// TIA Portal project "Endüstriyel Kapı" (V17)

(* hardware
DEVICE "S71500/ET200MP-Station_1"  S7-1500 station
   slot 0: "Profilschiene_0"  6ES7 590-1***0-0AA0
   slot 1: "PLC_1"  CPU 1511-1 PN  6ES7 511-1AK00-0AB0  V1.8
   slot 2: "AI 8xU/I/RTD/TC ST_1"  AI 8xU/I/RTD/TC ST  6ES7 531-7KF00-0AB0  V2.0
   slot 3: "AI 8xU/I/RTD/TC ST_2"  AI 8xU/I/RTD/TC ST  6ES7 531-7KF00-0AB0  V2.0
   slot 4: "AI 8xU/I/RTD/TC ST_3"  AI 8xU/I/RTD/TC ST  6ES7 531-7KF00-0AB0  V2.0
   slot 5: "AI 8xU/I/RTD/TC ST_4"  AI 8xU/I/RTD/TC ST  6ES7 531-7KF00-0AB0  V2.0
   slot 6: "DI 16x24VDC BA_1"  DI 16x24VDC BA  6ES7 521-1BH10-0AA0  V1.0
*)

// ===== PLC "PLC_1"  CPU 1511-1 PN =====

VAR_GLOBAL   // PLC tag table "Standard-Variablentabelle"
   "AÇMA (MÜHÜRLÜ)" AT %E0.0 : Bool;
   "AÇMA (KESİK)" AT %E0.1 : Bool;
   "KAPAMA (MÜHÜRLÜ)" AT %I0.2 : Bool;
   "KAPAMA (KESİK)" AT %I0.3 : Bool;
   "YAKINLIK SENSÖRÜ" AT %I0.4 : Bool;
   "KAPI AÇIK SENSÖR" AT %I0.5 : Bool;
   "KAPI KAPALI SENSÖR" AT %I0.6 : Bool;
   "ACİL STOP" AT %I0.7 : Bool;
   "KAPI AÇMA" AT %Q0.0 : Bool;
   "KAPI KAPAMA" AT %Q0.1 : Bool;
   "UYARI IŞIK" AT %Q0.2 : Bool;
   "KAPI AÇMA Y.K" AT %M0.0 : Bool;
   "KAPI KAPAMA Y.K" AT %M0.1 : Bool;
END_VAR

// folder: System blocks/Program resources

DATA_BLOCK "T0"   // DB1
{ S7_Optimized_Access := 'TRUE' }
AUTHOR : Simatic
FAMILY : IEC
NAME : IEC_TMR
VERSION : 1.0
// stored: InstanceOfName IEC_TIMER
"IEC_TIMER"
BEGIN
END_DATA_BLOCK

// folder: (top level)

FUNCTION "MHJ-PLC-Lab-Function-S71500" : Void   // FC9000, SCL
{ S7_Optimized_Access := 'TRUE' }
VERSION : 0.1
   VAR_TEMP
      Value : Byte;
      ForCounter : Int;
   END_VAR
   VAR CONSTANT
      Value_01_DW : DWord := 16#1223_5486;
      Value_02_DW : DWord := 16#A6C9_D1F5;
   END_VAR
BEGIN

   #Value:=PEEK(area := 16#82,
        dbNumber := 0,
        byteOffset := 511);
   #Value := #Value + 1;

   POKE(area := 16#82,
        dbNumber := 0,
        byteOffset := 511,
        value := #Value);

   POKE(area := 16#82,
        dbNumber := 0,
        byteOffset := 1016,
        value := #Value_01_DW);
   POKE(area := 16#82,
        dbNumber := 0,
        byteOffset := 1020,
        value := #Value_02_DW);

   FOR #ForCounter := 0 TO 63 DO
       #Value:=PEEK(area := 16#1,
            dbNumber := 0,
            byteOffset := #ForCounter);
       POKE(area := 16#81,
            dbNumber := 0,
            byteOffset := #ForCounter,
            value := #Value);
   END_FOR;
   #Value := PEEK(area := 16#1,
                  dbNumber := 0,
                  byteOffset := 512);
   POKE(area := 16#82,
        dbNumber := 0,
        byteOffset := 512,
        value := #Value);
END_FUNCTION

ORGANIZATION_BLOCK "Main"   // OB1, LAD, ProgramCycle
TITLE = "Main Program Sweep (Cycle)"
{ S7_Optimized_Access := 'TRUE' }
VERSION : 0.1
   VAR_INPUT
      Initial_Call : Bool;   // Initial call of this OB
      Remanence : Bool;   // =True, if remanent data are available
   END_VAR
BEGIN

REGION Network 1
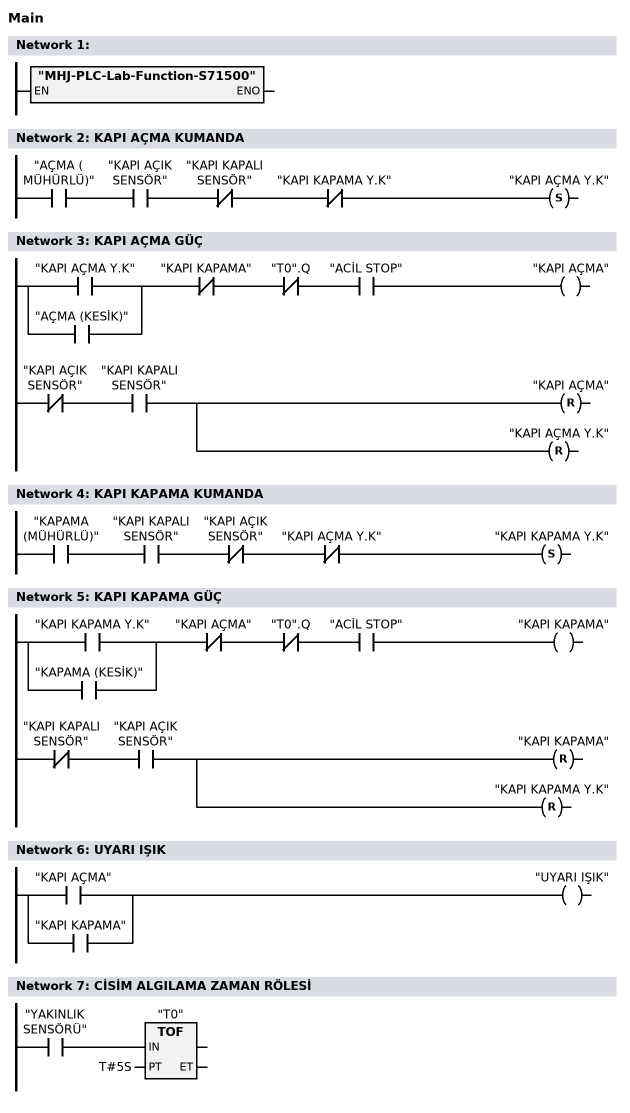
   RUNG wire#powerrail
      "MHJ-PLC-Lab-Function-S71500"()
   END_RUNG
   // the same network as SCL:
   "MHJ-PLC-Lab-Function-S71500"();
END_REGION

REGION Network 2: KAPI AÇMA KUMANDA
   RUNG wire#powerrail
      Contact( "AÇMA (MÜHÜRLÜ)" )
      Contact( "KAPI AÇIK SENSÖR" )
      I_Contact( "KAPI KAPALI SENSÖR" )
      I_Contact( "KAPI KAPAMA Y.K" )
      S_Coil( "KAPI AÇMA Y.K" )
   END_RUNG
   // the same network as SCL:
   IF "AÇMA (MÜHÜRLÜ)" AND "KAPI AÇIK SENSÖR" AND NOT "KAPI KAPALI SENSÖR" AND NOT "KAPI KAPAMA Y.K" THEN
       "KAPI AÇMA Y.K" := TRUE;
   END_IF;
END_REGION

REGION Network 3: KAPI AÇMA GÜÇ
   RUNG wire#powerrail
      Contact( "KAPI AÇMA Y.K" )
      wire#w1
      I_Contact( "KAPI KAPAMA" )
      I_Contact( "T0".Q )
      Contact( "ACİL STOP" )
      Coil( "KAPI AÇMA" )
   END_RUNG
   RUNG wire#powerrail
      Contact( "AÇMA (KESİK)" )
   END_RUNG wire#w1
   RUNG wire#powerrail
      I_Contact( "KAPI AÇIK SENSÖR" )
      Contact( "KAPI KAPALI SENSÖR" )
      wire#w2
      R_Coil( "KAPI AÇMA" )
   END_RUNG
   RUNG wire#w2
      R_Coil( "KAPI AÇMA Y.K" )
   END_RUNG
   // the same network as SCL:
   "KAPI AÇMA" := ("KAPI AÇMA Y.K" OR "AÇMA (KESİK)") AND NOT "KAPI KAPAMA" AND NOT "T0".Q AND "ACİL STOP";
   IF NOT "KAPI AÇIK SENSÖR" AND "KAPI KAPALI SENSÖR" THEN
       "KAPI AÇMA" := FALSE;
       "KAPI AÇMA Y.K" := FALSE;
   END_IF;
END_REGION

REGION Network 4: KAPI KAPAMA KUMANDA
   RUNG wire#powerrail
      Contact( "KAPAMA (MÜHÜRLÜ)" )
      Contact( "KAPI KAPALI SENSÖR" )
      I_Contact( "KAPI AÇIK SENSÖR" )
      I_Contact( "KAPI AÇMA Y.K" )
      S_Coil( "KAPI KAPAMA Y.K" )
   END_RUNG
   // the same network as SCL:
   IF "KAPAMA (MÜHÜRLÜ)" AND "KAPI KAPALI SENSÖR" AND NOT "KAPI AÇIK SENSÖR" AND NOT "KAPI AÇMA Y.K" THEN
       "KAPI KAPAMA Y.K" := TRUE;
   END_IF;
END_REGION

REGION Network 5: KAPI KAPAMA GÜÇ
   RUNG wire#powerrail
      Contact( "KAPI KAPAMA Y.K" )
      wire#w1
      I_Contact( "KAPI AÇMA" )
      I_Contact( "T0".Q )
      Contact( "ACİL STOP" )
      Coil( "KAPI KAPAMA" )
   END_RUNG
   RUNG wire#powerrail
      Contact( "KAPAMA (KESİK)" )
   END_RUNG wire#w1
   RUNG wire#powerrail
      I_Contact( "KAPI KAPALI SENSÖR" )
      Contact( "KAPI AÇIK SENSÖR" )
      wire#w2
      R_Coil( "KAPI KAPAMA" )
   END_RUNG
   RUNG wire#w2
      R_Coil( "KAPI KAPAMA Y.K" )
   END_RUNG
   // the same network as SCL:
   "KAPI KAPAMA" := ("KAPI KAPAMA Y.K" OR "KAPAMA (KESİK)") AND NOT "KAPI AÇMA" AND NOT "T0".Q AND "ACİL STOP";
   IF NOT "KAPI KAPALI SENSÖR" AND "KAPI AÇIK SENSÖR" THEN
       "KAPI KAPAMA" := FALSE;
       "KAPI KAPAMA Y.K" := FALSE;
   END_IF;
END_REGION

REGION Network 6: UYARI IŞIK
   RUNG wire#powerrail
      Contact( "KAPI AÇMA" )
      wire#w1
      Coil( "UYARI IŞIK" )
   END_RUNG
   RUNG wire#powerrail
      Contact( "KAPI KAPAMA" )
   END_RUNG wire#w1
   // the same network as SCL:
   "UYARI IŞIK" := "KAPI AÇMA" OR "KAPI KAPAMA";
END_REGION

REGION Network 7: CİSİM ALGILAMA ZAMAN RÖLESİ
   "T0".TOF(IN := "YAKINLIK SENSÖRÜ", PT := T#5S);
END_REGION
END_ORGANIZATION_BLOCK